// TIA Portal V17 export
VAR_GLOBAL   // PLC tag table "AlveTestTable"
   MyMinimal AT %I0.7 : Bool;
   MyRemoveAttributes AT %I1.0 : Bool;   //    {ExternalAccessible false, ExternalVisible false, ExternalWritable false}
   MyMemory AT %M1.1 : Bool;
   MyOutput AT %Q1.2 : Bool;
END_VAR
